PROGRAM RunMotor
VAR
END_VAR

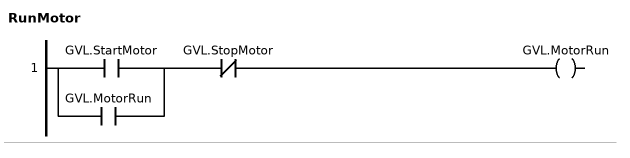
// NETWORK 1
GVL.MotorRun := (GVL.StartMotor OR GVL.MotorRun) AND NOT GVL.StopMotor;

END_PROGRAM

(* stored: Version 1.1.0.1, ProductVersion 3.1.4024.12
   POU RunMotor: Id {259652a1-9ecf-4c09-998d-63f3b033e923}, SpecialFunc None *)
